(* CoDeSys 2.3.9.28 project: Ex2.pro *)
(* Libraries: Standard.lib 27.1.09 11:27:38, Util.lib 27.1.09 11:27:38, IecSfc.lib*24.11.08 08:07:15, SysLibTime.lib*27.1.09 11:27:38, SysTaskInfo.lib 24.11.08 08:07:15, SYSLIBCALLBACK.LIB 27.1.09 11:27:38 *)

(* PLC configuration (modules and I/O channels)
Hexswitch AT %IB0 [HexSwitch] rotary switch 0 = STOP, 1-15 = RUN
8DI/8DO [CPX-8DI_8DO_Multi_I_O_module_1] node 0, in %IB4 out %QB0 {StringParam = 4,8,1,8,1; ByteParam = 7; ByteParam = 81; ByteParam = 0; ByteParam = 0; ByteParam = 0; ByteParam = 0; ByteParam = 0; IdleStateParam = 0; IdleModeParam = 255; IdleStateParam = 0; IdleModeParam = 255; IdleStateParam = 0; IdleModeParam = 255; IdleStateParam = 0; IdleModeParam = 255}
  AT %IB4 [ByteInput] -
  AT %QB0 [ByteOutput] -
8DI/8DO [CPX-8DI_8DO_Multi_I_O_module_1] node 1, in %IB8 out %QB4 {StringParam = 4,8,1,8,1; ByteParam = 7; ByteParam = 81; ByteParam = 0; ByteParam = 0; ByteParam = 0; ByteParam = 0; ByteParam = 0; IdleStateParam = 0; IdleModeParam = 255; IdleStateParam = 0; IdleModeParam = 255; IdleStateParam = 0; IdleModeParam = 255; IdleStateParam = 0; IdleModeParam = 255}
  AT %IB8 [ByteInput] -
  AT %QB4 [ByteOutput] -
*)

(* Global variable list: Global_Variables *)
VAR_GLOBAL

	START AT  %IX2.0 : BOOL;
	STOP AT  %IX2.1 : BOOL;
	S1 AT  %IX2.2 : BOOL;
	S2 AT  %IX2.3 : BOOL;
	S3 AT  %IX2.4 : BOOL;
	S4 AT  %IX2.5 : BOOL;

	L1 AT  %QX0.0 : BOOL;
	M1 AT  %QX0.1 : BOOL;
	M2 AT  %QX0.2 : BOOL;
	C1 AT  %QX0.3 : BOOL;
	C2 AT  %QX0.4 : BOOL;

END_VAR

(* POU PLC_PRG, LD *)
PROGRAM PLC_PRG
VAR
END_VAR
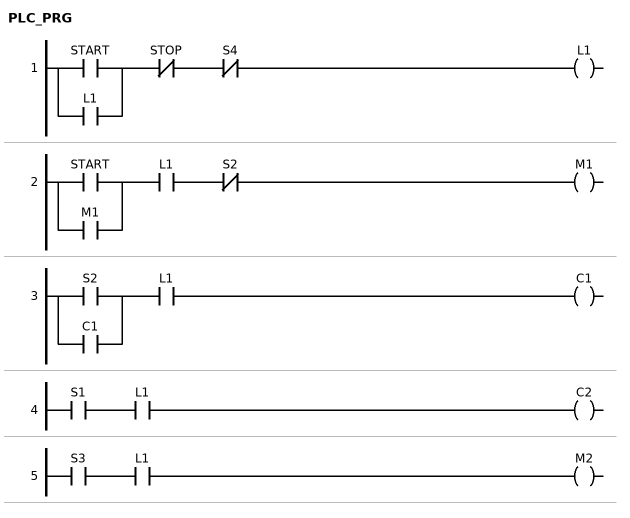
_LD_ (* Ladder Diagram *)
NETWORK 1
	{ [START] | [L1] } - [/STOP] - [/S4] --- (L1)
NETWORK 2
	{ [START] | [M1] } - [L1] - [/S2] --- (M1)
NETWORK 3
	{ [S2] | [C1] } - [L1] --- (C1)
NETWORK 4
	[S1] - [L1] --- (C2)
NETWORK 5
	[S3] - [L1] --- (M2)
_END_LD_
(* the same logic as Structured Text *)
(* Network 1 *)
L1 := (START OR L1) AND NOT STOP AND NOT S4;
(* Network 2 *)
M1 := (START OR M1) AND L1 AND NOT S2;
(* Network 3 *)
C1 := (S2 OR C1) AND L1;
(* Network 4 *)
C2 := S1 AND L1;
(* Network 5 *)
M2 := S3 AND L1;
END_PROGRAM
